TYPE OLSResult :
STRUCT
	m : LREAL := 0; // calculated linear regression slope
	b : LREAL := 0; // calculated linear regression intercept
	R2 : LREAL := 0; // R squared
	status : INT := 0; // 0 : OK; >0 : any failure
END_STRUCT
END_TYPE

(* stored: Version 1.1.0.1, ProductVersion 3.1.0.36
   DUT OLSResult: Id {e1694662-cd84-4ad8-928f-eea9230a6d2b} *)
